# EPICS alarm handler configuration: epics/epics_alh/alarms_list_Acnet.alhConfig
GROUP NULL Acnet

CHANNEL Acnet F:NM2D1
CHANNEL Acnet F:NM2V
CHANNEL Acnet F:NM2H
CHANNEL Acnet F:NM3S
CHANNEL Acnet F:NM4AN
CHANNEL Acnet F:NM2SEM
CHANNEL Acnet I:BEAM21
CHANNEL Acnet I:VFOUT
CHANNEL Acnet I:FTSDF
CHANNEL Acnet E:M3TGHM
CHANNEL Acnet E:M3TGHS
CHANNEL Acnet E:M3TGVM
CHANNEL Acnet E:M3TGVS
CHANNEL Acnet E:M3TGHI
CHANNEL Acnet E:M3TGHF
CHANNEL Acnet E:M3TGVI
CHANNEL Acnet E:M3TGVF
CHANNEL Acnet E:M2C2HM
CHANNEL Acnet E:M2C2HS
CHANNEL Acnet E:M2C2VM
CHANNEL Acnet E:M2C2VS
CHANNEL Acnet E:M2C2HI
CHANNEL Acnet E:M2C2HF
CHANNEL Acnet E:M2C2VI
CHANNEL Acnet E:M2C2VF
CHANNEL Acnet L:CBAR
CHANNEL Acnet S:KTEVTC
CHANNEL Acnet F:NM2ION
CHANNEL Acnet F:NM3ION
CHANNEL Acnet F:NM3RST
CHANNEL Acnet F:NM3RRT
CHANNEL Acnet F:NS2SUP
CHANNEL Acnet F:NS2RET
CHANNEL Acnet M:OUTTMP
CHANNEL Acnet F:E906BM
CHANNEL Acnet S:G2SEM
CHANNEL Acnet G:TURN13
CHANNEL Acnet G:BNCH13
CHANNEL Acnet G:NBSYD
CHANNEL Acnet S:N2N3EF
CHANNEL Acnet U:TODB25
CHANNEL Acnet S:MSEP1U
CHANNEL Acnet S:F1SEM
CHANNEL Acnet F:NM2Q1
CHANNEL Acnet F:NM2Q2
CHANNEL Acnet F:NS2FLO
CHANNEL Acnet F:NM3SEM
CHANNEL Acnet F:NS7DFP
CHANNEL Acnet G:RD3161
CHANNEL Acnet G:RD3162
CHANNEL Acnet F:MT6SC1
CHANNEL Acnet F:MC7SC1
CHANNEL Acnet F:MC1D
CHANNEL Acnet F:MW1W
